(* IEC 61131-3 sources: test/Class/SfcClass_Transition0, 1 file *)

(* ---- SfcClass_Transition0.st ---- *)
(*!
<Class
	Name               = "SfcClass_Transition0"
	Revision           = "0.0"
	RealtimeTask       = "false"
	CyclicTask         = "false"
	BackgroundTask     = "false"
	Sigmatek           = "false"
	OSInterface        = "false"
	HighPriority       = "false"
	Automatic          = "false"
	UpdateMode         = "Prescan"
	SharedCommandTable = "true"
	Objectsize         = "(284,120)">
	<Channels>
	</Channels>
	<Network Name="SfcClass_Transition0">
		<!-- List of Components in this network -->
		<Components>
			<Object
				Name       = "_base"
				Class      = "Sfc_Transition_Base"
				Position   = "(218,120)"
				Visualized = "false">
				<Channels>
					<Server Name="TransitionItf"/>
					<Client Name="GetParentPtr"/>
					<Client Name="NextStep"/>
					<Client Name="PrevStep"/>
				</Channels>
			</Object>
		</Components>
		<Comments>
		</Comments>
		<!-- List of Connections in this network -->
		<Connections>
			<Connection Source="this.TransitionItf" Destination="_base.TransitionItf" Vertices="(690,210),(518,210),"/>
			<Connection Source="_base.PrevStep" Destination="this.PrevStep" Vertices="(230,210),(38,210),"/>
			<Connection Source="_base.NextStep" Destination="this.NextStep" Vertices="(230,270),(38,270),"/>
			<Connection Source="_base.GetParentPtr" Destination="this.GetParentPtr" Vertices="(230,330),(38,330),"/>
		</Connections>
		<!-- Headerfiles -->
		<Options>
		</Options>
	</Network>
</Class>
*)
#pragma using Sfc_Transition_Base

SfcClass_Transition0 : CLASS
: Sfc_Transition_Base
	TYPE
	  pParentClsPtr : ^SfcClass;
	END_TYPE
  //Servers:
  //Clients:
  //Variables:
  //Functions:

	FUNCTION VIRTUAL Condition
		VAR_OUTPUT
			Result 	: DINT;
		END_VAR;
				//! <Function Name="OnReadInternalVariables" Hidden="true"/>
	FUNCTION VIRTUAL OnReadInternalVariables;
				//! <Function Name="OnWriteInternalVariables" Hidden="true"/>
	FUNCTION VIRTUAL OnWriteInternalVariables;
  //Tables:
	FUNCTION @STD
		VAR_OUTPUT
			ret_code	: CONFSTATES;
		END_VAR;
	FUNCTION GLOBAL TAB @CT_;
END_CLASS;

#pragma usingLtd SfcClass

FUNCTION VIRTUAL SfcClass_Transition0::OnReadInternalVariables

END_FUNCTION
FUNCTION VIRTUAL SfcClass_Transition0::OnWriteInternalVariables

END_FUNCTION

FUNCTION VIRTUAL SfcClass_Transition0::Condition
	VAR_OUTPUT
		Result 	: DINT;
	END_VAR

	Result := FALSE;

END_FUNCTION
